INTERFACE I_RpcHeaderAccessor

PROPERTY PUBLIC ContentType_Json : T_MAXSTRING
GET
END_GET
END_PROPERTY

METHOD PUBLIC TryGetAcceptResponseFormatFromRequest : BOOL
VAR_INPUT
	Request : I_Request;
	Destination : ANY;
END_VAR
END_METHOD

METHOD PUBLIC TryGetContentTypeFromRequest : BOOL
VAR_INPUT
	Request : I_Request;
	Destination : ANY;
END_VAR
END_METHOD

METHOD PUBLIC TryGetMethodNameFromRequest : BOOL
VAR_INPUT
	Request : I_Request;
	Destination : ANY;
END_VAR
END_METHOD

METHOD PUBLIC TryGetTypeFromRequest : BOOL
VAR_INPUT
	Request : I_Request;
	Destination : ANY;
END_VAR
END_METHOD

END_INTERFACE

(* stored: Version 1.1.0.1, ProductVersion 3.1.4024.12
   Itf I_RpcHeaderAccessor: Id {f1f1ac42-0ed5-4d02-93a4-3a3c64eacaab}
   Property ContentType_Json: Id {ae780374-5207-4c7b-8cac-f743608a01f8}
   Get Get: Id {60379507-d8ee-4101-8a76-49d4785ff62a}
   Method TryGetAcceptResponseFormatFromRequest: Id {97529f92-ea6c-4e19-af04-1f89e853f35f}
   Method TryGetContentTypeFromRequest: Id {39137155-f1f5-4510-8154-5d4e687fc0fb}
   Method TryGetMethodNameFromRequest: Id {37a464cc-0950-4ccb-a0a7-1c05e3c2ea92}
   Method TryGetTypeFromRequest: Id {ac6c1ba2-f2e7-46c2-a005-dc4916581629} *)
